GLOBALCONSTANTS logiBUS_DO (* logiBUS_DO constants *)
  (* Standard: 61499-1; Description: Copyright (c) 2024 HR Agrartechnik GmbH This program and the accompanying materials are made available under the terms of the Eclipse Public License 2.0 which is available at https://www.eclipse.org/legal/epl-2.0/ SPDX-License-Identifier: EPL-2.0 *)
  (* Version 1.0, 2024-01-25, Franz Höpfinger, HR Agrartechnik GmbH *)
  PACKAGE logiBUS::io::DQ;
  IMPORT eclipse4diac::core::TypeHash;
  VAR_GLOBAL CONSTANT
    Output_Q1 : logiBUS::io::DQ::logiBUS_DO_S := (Pin := 1);
    Output_Q2 : logiBUS::io::DQ::logiBUS_DO_S := (Pin := 2);
    Output_Q3 : logiBUS::io::DQ::logiBUS_DO_S := (Pin := 3);
    Output_Q4 : logiBUS::io::DQ::logiBUS_DO_S := (Pin := 4);
    Output_Q5 : logiBUS::io::DQ::logiBUS_DO_S := (Pin := 5);
    Output_Q6 : logiBUS::io::DQ::logiBUS_DO_S := (Pin := 6);
    Output_Q7 : logiBUS::io::DQ::logiBUS_DO_S := (Pin := 7);
    Output_Q8 : logiBUS::io::DQ::logiBUS_DO_S := (Pin := 8);
    Output_Q9 : logiBUS::io::DQ::logiBUS_DO_S := (Pin := 9);
    Output_Q10 : logiBUS::io::DQ::logiBUS_DO_S := (Pin := 10);
    Output_Q11 : logiBUS::io::DQ::logiBUS_DO_S := (Pin := 11);
    Output_Q12 : logiBUS::io::DQ::logiBUS_DO_S := (Pin := 12);
    Output_Q56 : logiBUS::io::DQ::logiBUS_DO_S := (Pin := 56);
    Output_Q78 : logiBUS::io::DQ::logiBUS_DO_S := (Pin := 78);
    Invalid : logiBUS::io::DQ::logiBUS_DO_S := (Pin := 255);
  END_VAR
END_GLOBALCONSTANTS
